{attribute 'GeneratedUsingTerminal: EJ1859-0000-0017'}
{attribute addProperty BoxType "EJ1859-0000-0017"}
{attribute addProperty Id "OutputAT %Q*BOOL1"}
{attribute addProperty CRC "1120571895"}
{attribute addProperty Size "1"}
TYPE Channel_42CA91F7 EXTENDS OutputBase_10CEE7DE :
STRUCT
	{attribute addProperty Name "Output"}
	Output AT %Q* : BOOL;
END_STRUCT
END_TYPE

(* stored: Version 1.2.0.0, ProductVersion 3.1.4024.9
   DUT Channel_42CA91F7: Id {dd44b68e-b621-4312-b47a-5dbc066a700b} *)
